// TIA Portal V17 export
// export: Created 2022-03-12T16:05:14.3241796Z, ExportSetting WithDefaults, DisplayName Totally Integrated Automation Portal, DisplayVersion V17, DisplayName TIA Portal Openness, DisplayVersion V17, DisplayName TIA Portal Version Control Interface, DisplayVersion V17, DisplayName STEP 7 Professional, DisplayVersion V17, DisplayName STEP 7 Safety, DisplayVersion V17, DisplayName WinCC Advanced / Unified PC, DisplayVersion V17
FUNCTION_BLOCK "UN_03_LineComm"   // FB31623, LAD
TITLE = UN_03_LineComm
{ S7_Optimized_Access := 'TRUE' }
AUTHOR : tech.team.motioncontrol@siemens.com
FAMILY : CPG
VERSION : 1.0
// Support: tech.team.motioncontrol@siemens.com
// Fax: +49 (0) 9131/98-1297
// stored: AutoNumber true, IsIECCheckEnabled false, IsRetainMemResEnabled false, MemoryReserve 100, SetENOAutomatically false, UDAEnableTagReadback false
   VAR
      instAlarmRemoteStop { ExternalAccessible := 'False'; ExternalVisible := 'False'; ExternalWritable := 'False'; S7_SetPoint := 'True'} : "CPG_Event";   // Remote Command - Stop
      instAlarmRemoteAbort { ExternalAccessible := 'False'; ExternalVisible := 'False'; ExternalWritable := 'False'; S7_SetPoint := 'True'} : "CPG_Event";   // Remote Command - Abort
      instAlarmRemoteSuspendBlocked { ExternalAccessible := 'False'; ExternalVisible := 'False'; ExternalWritable := 'False'; S7_SetPoint := 'True'} : "CPG_Event";   // Remote Command - Suspend (Blocked)
      instAlarmRemoteSuspendStarved { ExternalAccessible := 'False'; ExternalVisible := 'False'; ExternalWritable := 'False'; S7_SetPoint := 'True'} : "CPG_Event";   // Remote Command - Suspend (Starved)
      instAlarmRemoteHold { ExternalAccessible := 'False'; ExternalVisible := 'False'; ExternalWritable := 'False'; S7_SetPoint := 'True'} : "CPG_Event";   // Remote Command - Hold
      statRemoteSuspendCommand { ExternalAccessible := 'False'; ExternalVisible := 'False'; ExternalWritable := 'False'} : Bool;   // Remote Suspend Command is active (from remote station)
      statRemoteHoldCommand { ExternalAccessible := 'False'; ExternalVisible := 'False'; ExternalWritable := 'False'} : Bool;   // Remote Hold Command is active (from remote station)
   END_VAR
BEGIN

REGION Network 1: *** COMMUNICATION LOGIC ***
END_REGION

REGION Network 2: *** REMOTE COMMAND LOGIC ***
END_REGION

REGION Network 3: Remote Stop Command
   // "PackTags".Command.CntrlCmd = 3 (stop command value)
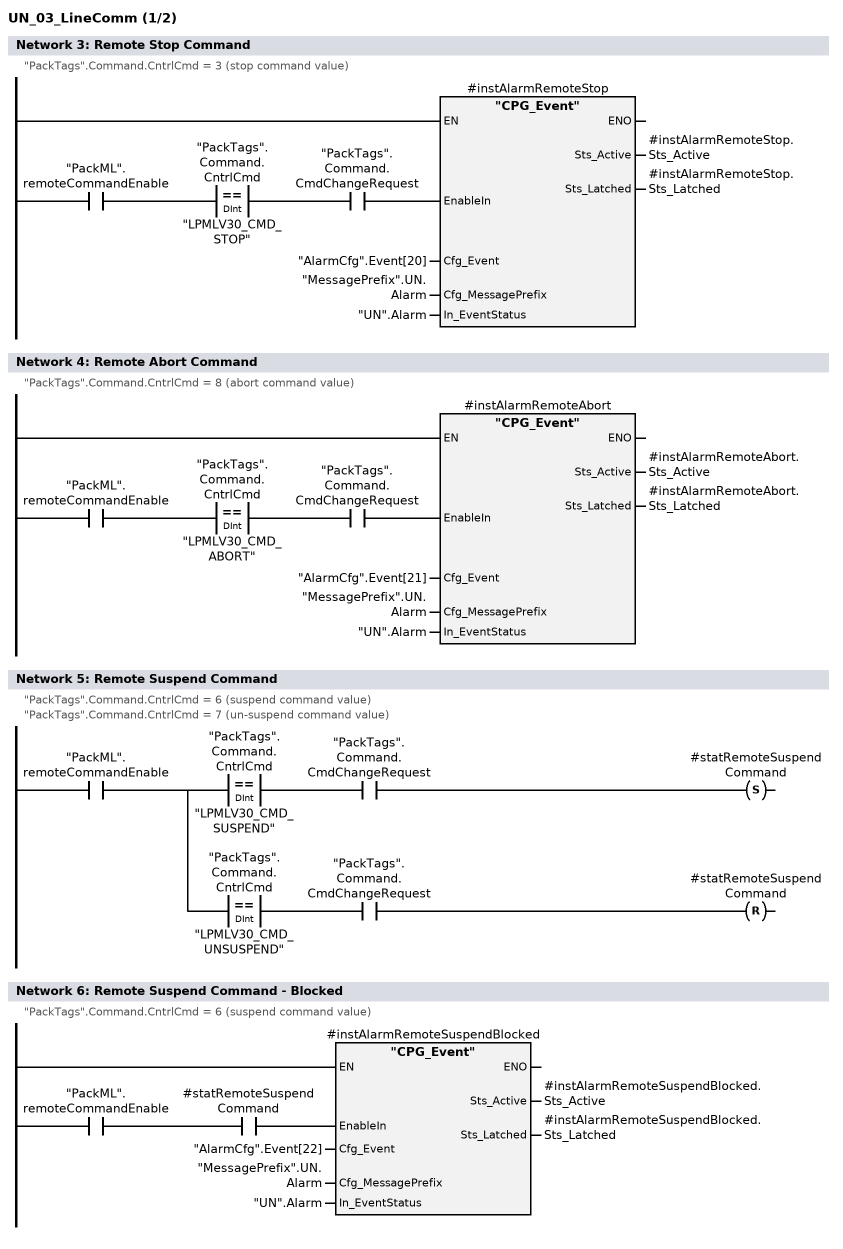
   RUNG wire#powerrail
      #instAlarmRemoteStop(EnableIn := wire#w1, Cfg_Event := "AlarmCfg".Event[20], Cfg_MessagePrefix := "MessagePrefix".UN.Alarm, In_EventStatus := "UN".Alarm, Sts_Active => #instAlarmRemoteStop.Sts_Active, Sts_Latched => #instAlarmRemoteStop.Sts_Latched)
   END_RUNG
   RUNG wire#powerrail
      Contact( "PackML".remoteCommandEnable )
      { S7_Templates := "SrcType := DInt" } EQ_Contact(in1 := "PackTags".Command.CntrlCmd, in2 := "LPMLV30_CMD_STOP")
      Contact( "PackTags".Command.CmdChangeRequest )
   END_RUNG wire#w1
   // the same network as SCL:
   #instAlarmRemoteStop(EnableIn := "PackML".remoteCommandEnable AND ("PackTags".Command.CntrlCmd = "LPMLV30_CMD_STOP") AND "PackTags".Command.CmdChangeRequest,   // "CPG_Event"
                        Cfg_Event := "AlarmCfg".Event[20],
                        Cfg_MessagePrefix := "MessagePrefix".UN.Alarm,
                        In_EventStatus := "UN".Alarm,
                        Sts_Active => #instAlarmRemoteStop.Sts_Active,
                        Sts_Latched => #instAlarmRemoteStop.Sts_Latched);
END_REGION

REGION Network 4: Remote Abort Command
   // "PackTags".Command.CntrlCmd = 8 (abort command value)
   RUNG wire#powerrail
      #instAlarmRemoteAbort(EnableIn := wire#w1, Cfg_Event := "AlarmCfg".Event[21], Cfg_MessagePrefix := "MessagePrefix".UN.Alarm, In_EventStatus := "UN".Alarm, Sts_Active => #instAlarmRemoteAbort.Sts_Active, Sts_Latched => #instAlarmRemoteAbort.Sts_Latched)
   END_RUNG
   RUNG wire#powerrail
      Contact( "PackML".remoteCommandEnable )
      { S7_Templates := "SrcType := DInt" } EQ_Contact(in1 := "PackTags".Command.CntrlCmd, in2 := "LPMLV30_CMD_ABORT")
      Contact( "PackTags".Command.CmdChangeRequest )
   END_RUNG wire#w1
   // the same network as SCL:
   #instAlarmRemoteAbort(EnableIn := "PackML".remoteCommandEnable AND ("PackTags".Command.CntrlCmd = "LPMLV30_CMD_ABORT") AND "PackTags".Command.CmdChangeRequest,   // "CPG_Event"
                         Cfg_Event := "AlarmCfg".Event[21],
                         Cfg_MessagePrefix := "MessagePrefix".UN.Alarm,
                         In_EventStatus := "UN".Alarm,
                         Sts_Active => #instAlarmRemoteAbort.Sts_Active,
                         Sts_Latched => #instAlarmRemoteAbort.Sts_Latched);
END_REGION

REGION Network 5: Remote Suspend Command
   // "PackTags".Command.CntrlCmd = 6 (suspend command value)
   // "PackTags".Command.CntrlCmd = 7 (un-suspend command value)
   RUNG wire#powerrail
      Contact( "PackML".remoteCommandEnable )
      wire#w1
      { S7_Templates := "SrcType := DInt" } EQ_Contact(in1 := "PackTags".Command.CntrlCmd, in2 := "LPMLV30_CMD_SUSPEND")
      Contact( "PackTags".Command.CmdChangeRequest )
      S_Coil( #statRemoteSuspendCommand )
   END_RUNG
   RUNG wire#w1
      { S7_Templates := "SrcType := DInt" } EQ_Contact(in1 := "PackTags".Command.CntrlCmd, in2 := "LPMLV30_CMD_UNSUSPEND")
      Contact( "PackTags".Command.CmdChangeRequest )
      R_Coil( #statRemoteSuspendCommand )
   END_RUNG
   // the same network as SCL:
   IF "PackML".remoteCommandEnable AND ("PackTags".Command.CntrlCmd = "LPMLV30_CMD_SUSPEND") AND "PackTags".Command.CmdChangeRequest THEN
       #statRemoteSuspendCommand := TRUE;
   END_IF;
   IF "PackML".remoteCommandEnable AND ("PackTags".Command.CntrlCmd = "LPMLV30_CMD_UNSUSPEND") AND "PackTags".Command.CmdChangeRequest THEN
       #statRemoteSuspendCommand := FALSE;
   END_IF;
END_REGION

REGION Network 6: Remote Suspend Command - Blocked
   // "PackTags".Command.CntrlCmd = 6 (suspend command value)
   RUNG wire#powerrail
      #instAlarmRemoteSuspendBlocked(EnableIn := wire#w1, Cfg_Event := "AlarmCfg".Event[22], Cfg_MessagePrefix := "MessagePrefix".UN.Alarm, In_EventStatus := "UN".Alarm, Sts_Active => #instAlarmRemoteSuspendBlocked.Sts_Active, Sts_Latched => #instAlarmRemoteSuspendBlocked.Sts_Latched)
   END_RUNG
   RUNG wire#powerrail
      Contact( "PackML".remoteCommandEnable )
      Contact( #statRemoteSuspendCommand )
   END_RUNG wire#w1
   // the same network as SCL:
   #instAlarmRemoteSuspendBlocked(EnableIn := "PackML".remoteCommandEnable AND #statRemoteSuspendCommand,   // "CPG_Event"
                           Cfg_Event := "AlarmCfg".Event[22],
                           Cfg_MessagePrefix := "MessagePrefix".UN.Alarm,
                           In_EventStatus := "UN".Alarm,
                           Sts_Active => #instAlarmRemoteSuspendBlocked.Sts_Active,
                           Sts_Latched => #instAlarmRemoteSuspendBlocked.Sts_Latched);
END_REGION

REGION Network 7: Remote Suspend Command - Starved
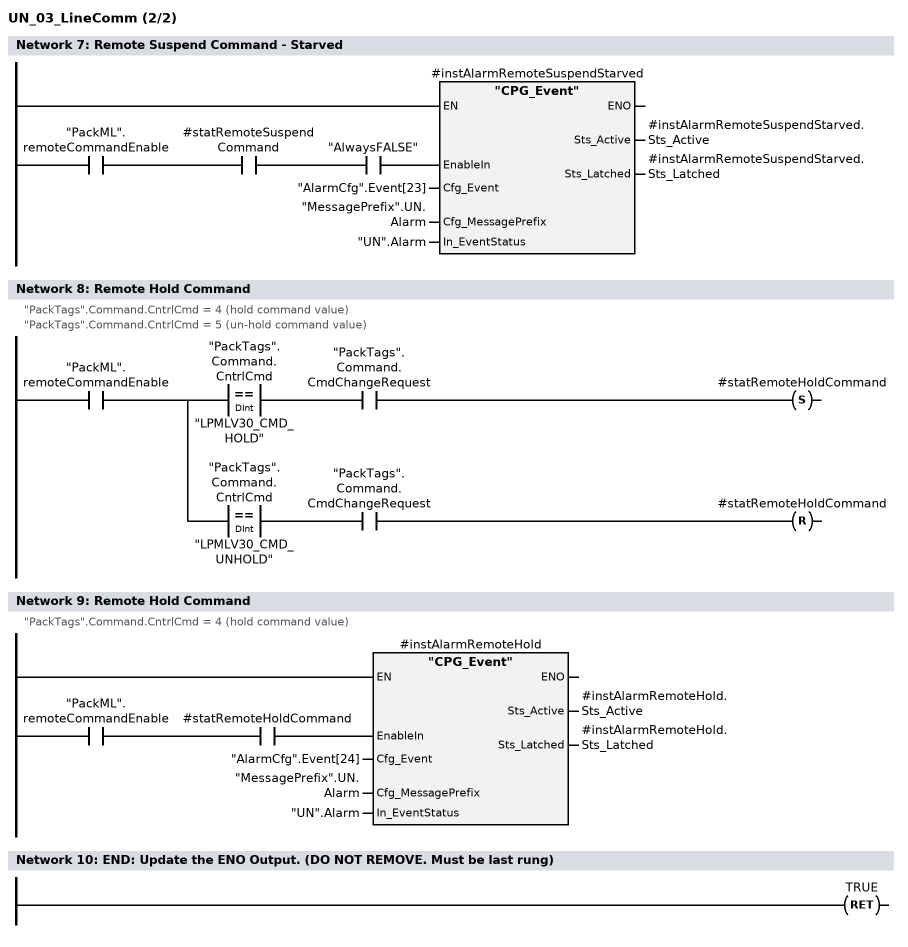
   RUNG wire#powerrail
      #instAlarmRemoteSuspendStarved(EnableIn := wire#w1, Cfg_Event := "AlarmCfg".Event[23], Cfg_MessagePrefix := "MessagePrefix".UN.Alarm, In_EventStatus := "UN".Alarm, Sts_Active => #instAlarmRemoteSuspendStarved.Sts_Active, Sts_Latched => #instAlarmRemoteSuspendStarved.Sts_Latched)
   END_RUNG
   RUNG wire#powerrail
      Contact( "PackML".remoteCommandEnable )
      Contact( #statRemoteSuspendCommand )
      Contact( "AlwaysFALSE" )
   END_RUNG wire#w1
   // the same network as SCL:
   #instAlarmRemoteSuspendStarved(EnableIn := "PackML".remoteCommandEnable AND #statRemoteSuspendCommand AND "AlwaysFALSE",   // "CPG_Event"
                           Cfg_Event := "AlarmCfg".Event[23],
                           Cfg_MessagePrefix := "MessagePrefix".UN.Alarm,
                           In_EventStatus := "UN".Alarm,
                           Sts_Active => #instAlarmRemoteSuspendStarved.Sts_Active,
                           Sts_Latched => #instAlarmRemoteSuspendStarved.Sts_Latched);
END_REGION

REGION Network 8: Remote Hold Command
   // "PackTags".Command.CntrlCmd = 4 (hold command value)
   // "PackTags".Command.CntrlCmd = 5 (un-hold command value)
   RUNG wire#powerrail
      Contact( "PackML".remoteCommandEnable )
      wire#w1
      { S7_Templates := "SrcType := DInt" } EQ_Contact(in1 := "PackTags".Command.CntrlCmd, in2 := "LPMLV30_CMD_HOLD")
      Contact( "PackTags".Command.CmdChangeRequest )
      S_Coil( #statRemoteHoldCommand )
   END_RUNG
   RUNG wire#w1
      { S7_Templates := "SrcType := DInt" } EQ_Contact(in1 := "PackTags".Command.CntrlCmd, in2 := "LPMLV30_CMD_UNHOLD")
      Contact( "PackTags".Command.CmdChangeRequest )
      R_Coil( #statRemoteHoldCommand )
   END_RUNG
   // the same network as SCL:
   IF "PackML".remoteCommandEnable AND ("PackTags".Command.CntrlCmd = "LPMLV30_CMD_HOLD") AND "PackTags".Command.CmdChangeRequest THEN
       #statRemoteHoldCommand := TRUE;
   END_IF;
   IF "PackML".remoteCommandEnable AND ("PackTags".Command.CntrlCmd = "LPMLV30_CMD_UNHOLD") AND "PackTags".Command.CmdChangeRequest THEN
       #statRemoteHoldCommand := FALSE;
   END_IF;
END_REGION

REGION Network 9: Remote Hold Command
   // "PackTags".Command.CntrlCmd = 4 (hold command value)
   RUNG wire#powerrail
      #instAlarmRemoteHold(EnableIn := wire#w1, Cfg_Event := "AlarmCfg".Event[24], Cfg_MessagePrefix := "MessagePrefix".UN.Alarm, In_EventStatus := "UN".Alarm, Sts_Active => #instAlarmRemoteHold.Sts_Active, Sts_Latched => #instAlarmRemoteHold.Sts_Latched)
   END_RUNG
   RUNG wire#powerrail
      Contact( "PackML".remoteCommandEnable )
      Contact( #statRemoteHoldCommand )
   END_RUNG wire#w1
   // the same network as SCL:
   #instAlarmRemoteHold(EnableIn := "PackML".remoteCommandEnable AND #statRemoteHoldCommand,   // "CPG_Event"
                        Cfg_Event := "AlarmCfg".Event[24],
                        Cfg_MessagePrefix := "MessagePrefix".UN.Alarm,
                        In_EventStatus := "UN".Alarm,
                        Sts_Active => #instAlarmRemoteHold.Sts_Active,
                        Sts_Latched => #instAlarmRemoteHold.Sts_Latched);
END_REGION

REGION Network 10: END: Update the ENO Output. (DO NOT REMOVE. Must be last rung)
   RUNG wire#powerrail
      ReturnCoil( TRUE )
   END_RUNG
   // the same network as SCL:
   ENO := TRUE;
   RETURN;
END_REGION
END_FUNCTION_BLOCK
